{attribute 'obsolete' := 'Use E_EpicsMotorCmd'}
TYPE ENUM_EpicsMotorCmd : E_EpicsMotorCmd; END_TYPE

(* stored: Version 1.1.0.1
   DUT ENUM_EpicsMotorCmd: Id {1155ba19-87b2-4fb1-82f5-6bdaff163e77} *)
